TYPE ST_TIME_PROPORTIONAL_THERMOSTAT_HMI :
STRUCT
	settings:	ST_TIME_PROPORTIONAL_THERMOSTAT_SETTINGS;
	state:		ST_TIME_PROPORTIONAL_THERMOSTAT_STATE;
END_STRUCT
END_TYPE

(* stored: Version 1.1.0.1
   DUT ST_TIME_PROPORTIONAL_THERMOSTAT_HMI: Id {2eb7048d-a44d-4e22-93a9-556bbba323a5} *)
